FUNCTION cholsl : INT
VAR_IN_OUT
	A:ARRAY[*,*] OF LREAL;
	aa:ARRAY[*,*] OF LREAL;
	p:ARRAY[*,*] OF LREAL;

END_VAR
VAR_INPUT
		n:SINT;
END_VAR
VAR
 i,j,k:SINT;
 sum:LREAL;
END_VAR

 IF (choldcsl((A),(aa),(p),n)=1) THEN
	cholsl:= 1;
END_IF
    FOR i := 0 TO n DO
        FOR j := i + 1  TO n DO 
            aa[i,j] := 0.0;
        END_FOR
    END_FOR
	
    FOR i := 0 TO n DO 
        aa[i,i] := aa[i,i] *aa[i,i];
        FOR k := i + 1 TO n DO 
            aa[i,i] :=  aa[i,i] + aa[k,i] * aa[k,i];
		END_FOR
        FOR j := i + 1 TO n DO 
            FOR k := j TO  n DO
                aa[i,j] := aa[i,j]+ aa[k,i] * aa[k,j];
            END_FOR
        END_FOR
    END_FOR
    FOR i := 0 TO n DO
        FOR j := 0 TO i DO
            aa[i,j] := aa[j,i];
        END_FOR
    END_FOR

    cholsl:= 0;

END_FUNCTION

(* stored: Version 1.1.0.1, ProductVersion 3.1.4024.12
   POU cholsl: Id {906897ee-9a80-4bfe-b6ec-bfcf0eefd7d0}, SpecialFunc None *)
